{attribute 'qualified_only'}
{attribute 'strict'}
TYPE eTcoRoboticsStopType : (
    Soft := 10,
    Quick := 20
);
END_TYPE

(* stored: Version 1.1.0.1, ProductVersion 3.1.4024.12
   DUT eTcoRoboticsStopType: Id {91ea8bd6-7351-4932-acb5-9f53f4835f9e} *)
